FUNCTION FC_Add : WORD
VAR_INPUT
	a :WORD;
	b :WORD;
END_VAR
VAR
END_VAR

FC_Add := a+b;

END_FUNCTION

(* stored: Version 1.1.0.1
   POU FC_Add: Id {5ab2304d-3d82-4d00-b605-b47bcc588cfb}, SpecialFunc None *)
